// TwinCAT 3 PLC project Sample
// ProgramVersion: 3.1.4020.2
// libraries:
//   MyLibrary01, * (MyCompany)
//   Tc2_Standard, * (Beckhoff Automation GmbH)
//   Tc2_System, * (Beckhoff Automation GmbH)
//   Tc3_Module, * (Beckhoff Automation GmbH)
// project tree:
//   GVLs/ GVL01.TcGVL
//   / PlcTask.TcTTO (not stored)
//   POUs/ FB_MyFoo.TcPOU, MAIN.TcPOU
// (motion and I/O tree: see PLC project library01)
// real-time tasks:
//   TASK PlcTask: cycle T#10ms, priority 20, ADS port 350

// ---- GVLs/GVL01.TcGVL
VAR_GLOBAL
	var01		:	INT;
END_VAR

// ---- POUs/FB_MyFoo.TcPOU
FUNCTION_BLOCK PUBLIC FB_MyFoo EXTENDS MyNamespace01.FB_Foo IMPLEMENTS MyNamespace01.I_Foo
VAR_INPUT
END_VAR
VAR_OUTPUT
END_VAR
VAR
END_VAR

{warning 'add method implementation'}
METHOD DoSomething : BOOL
END_METHOD

END_FUNCTION_BLOCK

// ---- POUs/MAIN.TcPOU
PROGRAM MAIN
VAR
	var01		:	INT;
END_VAR

MyNamespace01.GVL01.var01 := 1;		// global variable of the GVL of the library
GVL01.var01 := 2;					// global variable of the local GVL
var01 := 3;							// local variable

END_PROGRAM
